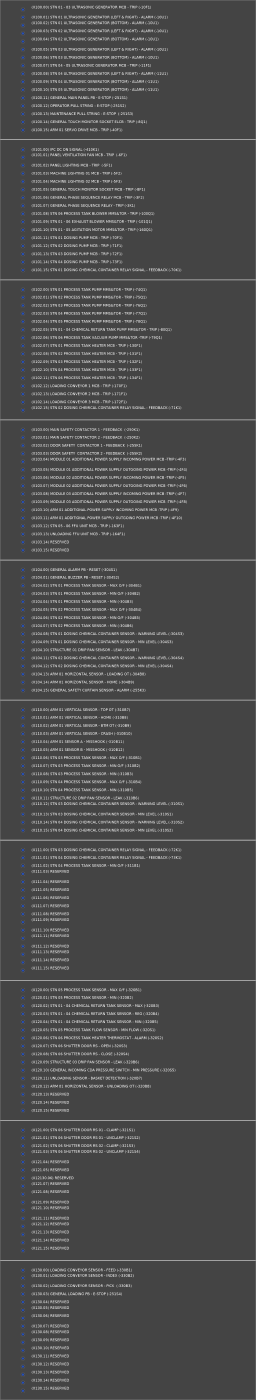
VISUALIZATION Popup_IOinput  // 733x3998
    Rectangle (0,0 733x398)
    Label (87,15 625x24), "(X100.00) STN 01 - 03 ULTRASONIC GENERATOR MCB - TRIP (-10F1)"
    Lamp1 (58,20 15x15), variable: ARbDI[eX10000_Stn01_03UltrasonicGeneratorMcb_Trip], style: Lamp-Lamp1-Blue
    Label (87,37 625x24), "(X100.01) STN 01 ULTRASONIC GENERATOR (LEFT & RIGHT) - ALARM (-10U1)"
    Lamp1 (58,42 15x15), variable: ARbDI[eX10001_Stn01UltrasonicGeneratorLeftRight_Alarm], style: Lamp-Lamp1-Blue
    Label (87,83 625x24), "(X100.03) STN 02 ULTRASONIC GENERATOR (LEFT & RIGHT) - ALARM (-10U1)"
    Lamp1 (58,88 15x15), variable: ARbDI[eX10003_Stn02UltrasonicGeneratorLeftRight_Alarm], style: Lamp-Lamp1-Blue
    Label (87,60 625x24), "(X100.02) STN 01 ULTRASONIC GENERATOR (BOTTOM) - ALARM (-10U1)"
    Lamp1 (58,65 15x15), variable: ARbDI[eX10002_Stn01UltrasonicGeneratorBottom_Alarm], style: Lamp-Lamp1-Blue
    Label (87,175 625x24), "(X100.07) STN 04 - 05 ULTRASONIC GENERATOR MCB - TRIP (-11F1)"
    Lamp1 (58,180 15x15), variable: ARbDI[eX10007_Stn04_05UltrasonicGeneratorMcb_Trip], style: Lamp-Lamp1-Blue
    Label (87,106 625x24), "(X100.04) STN 02 ULTRASONIC GENERATOR (BOTTOM) - ALARM (-10U1)"
    Lamp1 (58,111 15x15), variable: ARbDI[eX10004_Stn02UltrasonicGeneratorBottom_Alarm], style: Lamp-Lamp1-Blue
    Label (87,129 625x24), "(X100.05) STN 03 ULTRASONIC GENERATOR (LEFT & RIGHT) - ALARM (-10U1)"
    Lamp1 (58,134 15x15), variable: ARbDI[eX10005_Stn03UltrasonicGeneratorLeftRight_Alarm], style: Lamp-Lamp1-Blue
    Label (87,152 625x24), "(X100.06) STN 03 ULTRASONIC GENERATOR (BOTTOM) - ALARM (-10U1)"
    Lamp1 (58,157 15x15), variable: ARbDI[eX10006_Stn03UltrasonicGeneratorBottom_Alarm], style: Lamp-Lamp1-Blue
    Label (87,359 625x24), "(X100.15) ARM 01 SERVO DRIVE MCB - TRIP (-40F1)"
    Lamp1 (58,364 15x15), variable: ARbDI[eX10015_Arm01ServoDriveMcb_Trip], style: Lamp-Lamp1-Blue
    Label (87,198 625x24), "(X100.08) STN 04 ULTRASONIC GENERATOR (LEFT & RIGHT) - ALARM (-11U1)"
    Lamp1 (58,203 15x15), variable: ARbDI[eX10008_Stn04UltrasonicGeneratorLeftRight_Alarm], style: Lamp-Lamp1-Blue
    Label (87,221 625x24), "(X100.09) STN 04 ULTRASONIC GENERATOR (BOTTOM) - ALARM (-11U1)"
    Lamp1 (58,226 15x15), variable: ARbDI[eX10009_Stn04UltrasonicGeneratorBottom_Alarm], style: Lamp-Lamp1-Blue
    Label (87,267 625x24), "(X100.11) GENERAL MAIN PANEL PB - E-STOP (-251S1)"
    Lamp1 (58,272 15x15), variable: ARbDI[eX10011_GeneralMainPanelPb_E_Stop], style: Lamp-Lamp1-Blue
    Label (87,244 625x24), "(X100.10) STN 05 ULTRASONIC GENERATOR (BOTTOM) - ALARM (-11U1)"
    Lamp1 (58,249 15x15), variable: ARbDI[eX10010_Stn05UltrasonicGeneratorBottom_Alarm], style: Lamp-Lamp1-Blue
    Label (87,290 625x24), "(X100.12) OPERATOR PULL STRING - E-STOP (-251S2)"
    Lamp1 (58,295 15x15), variable: ARbDI[eX10012_OperatorPullString_E_Stop], style: Lamp-Lamp1-Blue
    Label (87,313 625x24), "(X100.13) MAINTENANCE PULL STRING - E-STOP (-251S3)"
    Lamp1 (58,318 15x15), variable: ARbDI[eX10013_MaintenancePullString_E_Stop], style: Lamp-Lamp1-Blue
    Label (87,336 625x24), "(X100.14) GENERAL TOUCH MONITOR SOCKET ELCB - TRIP (-8Q1)"
    Lamp1 (58,341 15x15), variable: ARbDI[eX10014_GeneralTouchMonitorSocketElcb_Trip], style: Lamp-Lamp1-Blue
    Rectangle (0,400 733x398)
    Label (87,415 625x24), "(X101.00) IPC DC ON SIGNAL (-410K1)"
    Lamp1 (58,420 15x15), variable: ARbDI[eX10100_IpcDcOnSignal], style: Lamp-Lamp1-Blue
    Label (87,437 625x24), "(X101.01) PANEL VENTILATION FAN MCB - TRIP (-6F1)"
    Lamp1 (58,442 15x15), variable: ARbDI[eX10101_PanelVentilationFanMcb_Trip], style: Lamp-Lamp1-Blue
    Label (87,483 625x24), "(X101.03) MACHINE LIGHTING 01 MCB - TRIP (-5F2)"
    Lamp1 (58,488 15x15), variable: ARbDI[eX10103_MachineLighting01Mcb_Trip], style: Lamp-Lamp1-Blue
    Label (87,460 625x24), "(X101.02) PANEL LIGHTING MCB - TRIP (-5F1)"
    Lamp1 (58,465 15x15), variable: ARbDI[eX10102_PanelLightingMcb_Trip], style: Lamp-Lamp1-Blue
    Label (87,575 625x24), "(X101.07) GENERAL PHASE SEQUENCE RELAY - TRIP (-3K1)"
    Lamp1 (58,580 15x15), variable: ARbDI[eX10107_GeneralPhaseSequenceRelay_Trip], style: Lamp-Lamp1-Blue
    Label (87,506 625x24), "(X101.04) MACHINE LIGHTING 02 MCB - TRIP (-5F3)"
    Lamp1 (58,511 15x15), variable: ARbDI[eX10104_MachineLighting02Mcb_Trip], style: Lamp-Lamp1-Blue
    Label (87,529 625x24), "(X101.05) GENERAL TOUCH MONITOR SOCKET MCB - TRIP (-8F1)"
    Lamp1 (58,534 15x15), variable: ARbDI[eX10105_GeneralTouchMonitorSocketMcb_Trip], style: Lamp-Lamp1-Blue
    Label (87,552 625x24), "(X101.06) GENERAL PHASE SEQUENCE RELAY MCB - TRIP (-3F2)"
    Lamp1 (58,557 15x15), variable: ARbDI[eX10106_GeneralPhaseSequenceRelayMcb_Trip], style: Lamp-Lamp1-Blue
    Label (87,759 625x24), "(X101.15) STN 01 DOSING CHEMICAL CONTAINER RELAY SIGNAL - FEEDBACK (-70K1)"
    Lamp1 (58,764 15x15), variable: ARbDI[eX10115_Stn01DosingChemicalContainerRelaySignal_Feedback], style: Lamp-Lamp1-Blue
    Label (87,598 625x24), "(X101.08) STN 06 PROCESS TANK BLOWER MMS&TOR - TRIP (-100Q1)"
    Lamp1 (58,603 15x15), variable: ARbDI[eX10108_Stn06ProcessTankBlowerMms_Tor_Trip], style: Lamp-Lamp1-Blue
    Label (87,621 625x24), "(X101.09) STN 01 - 06 EXHAUST BLOWER MMS&TOR - TRIP (-101Q1)"
    Lamp1 (58,626 15x15), variable: ARbDI[eX10109_Stn01_06ExhaustBlowerMms_Tor_Trip], style: Lamp-Lamp1-Blue
    Label (87,667 625x24), "(X101.11) STN 01 DOSING PUMP MCB - TRIP (-70F1)"
    Lamp1 (58,672 15x15), variable: ARbDI[eX10111_Stn01DosingPumpMcb_Trip], style: Lamp-Lamp1-Blue
    Label (87,644 625x24), "(X101.10) STN 01 - 05 AGITATION MOTOR MMS&TOR - TRIP (-160Q1)"
    Lamp1 (58,649 15x15), variable: ARbDI[eX10110_Stn01_05AgitationMotorMms_Tor_Trip], style: Lamp-Lamp1-Blue
    Label (87,690 625x24), "(X101.12) STN 02 DOSING PUMP MCB - TRIP (-71F1)"
    Lamp1 (58,695 15x15), variable: ARbDI[eX10112_Stn02DosingPumpMcb_Trip], style: Lamp-Lamp1-Blue
    Label (87,713 625x24), "(X101.13) STN 03 DOSING PUMP MCB - TRIP (-72F1)"
    Lamp1 (58,718 15x15), variable: ARbDI[eX10113_Stn03DosingPumpMcb_Trip], style: Lamp-Lamp1-Blue
    Label (87,736 625x24), "(X101.14) STN 04 DOSING PUMP MCB - TRIP (-73F1)"
    Lamp1 (58,741 15x15), variable: ARbDI[eX10114_Stn04DosingPumpMcb_Trip], style: Lamp-Lamp1-Blue
    Rectangle (0,800 733x398)
    Label (87,815 642x24), "(X102.00) STN 01 PROCESS TANK PUMP MMS&TOR - TRIP (-74Q1)"
    Lamp1 (58,820 15x15), variable: ARbDI[eX10200_Stn01ProcessTankPumpMms_Tor_Trip], style: Lamp-Lamp1-Blue
    Label (87,837 641x24), "(X102.01) STN 02 PROCESS TANK PUMP MMS&TOR - TRIP (-75Q1)"
    Lamp1 (58,842 15x15), variable: ARbDI[eX10201_Stn02ProcessTankPumpMms_Tor_Trip], style: Lamp-Lamp1-Blue
    Label (87,883 641x24), "(X102.03) STN 04 PROCESS TANK PUMP MMS&TOR - TRIP (-77Q1)"
    Lamp1 (58,888 15x15), variable: ARbDI[eX10203_Stn04ProcessTankPumpMms_Tor_Trip], style: Lamp-Lamp1-Blue
    Label (87,860 643x24), "(X102.02) STN 03 PROCESS TANK PUMP MMS&TOR - TRIP (-76Q1)"
    Lamp1 (58,865 15x15), variable: ARbDI[eX10202_Stn03ProcessTankPumpMms_Tor_Trip], style: Lamp-Lamp1-Blue
    Label (87,975 625x24), "(X102.07) STN 01 PROCESS TANK HEATER MCB - TRIP (-130F1)"
    Lamp1 (58,980 15x15), variable: ARbDI[eX10207_Stn01ProcessTankHeaterMcb_Trip], style: Lamp-Lamp1-Blue
    Label (87,906 641x24), "(X102.04) STN 05 PROCESS TANK PUMP MMS&TOR - TRIP (-78Q1)"
    Lamp1 (58,911 15x15), variable: ARbDI[eX10204_Stn05ProcessTankPumpMms_Tor_Trip], style: Lamp-Lamp1-Blue
    Label (87,929 642x24), "(X102.05) STN 01 - 04 CHEMICAL RETURN TANK PUMP MMS&TOR - TRIP (-80Q1)"
    Lamp1 (58,934 15x15), variable: ARbDI[eX10205_Stn01_04ChemicalReturnTankPumpMms_Tor_Trip], style: Lamp-Lamp1-Blue
    Label (87,952 642x24), "(X102.06) STN 06 PROCESS TANK VACUUM PUMP MMS&TOR -TRIP (-79Q1)"
    Lamp1 (58,957 15x15), variable: ARbDI[eX10206_Stn06ProcessTankVacuumPumpMms_Tor_Trip], style: Lamp-Lamp1-Blue
    Label (87,1159 625x24), "(X102.15) STN 02 DOSING CHEMICAL CONTAINER RELAY SIGNAL - FEEDBACK (-71K1)"
    Lamp1 (58,1164 15x15), variable: ARbDI[eX10215_Stn02DosingChemicalContainerRelaySignal_Feedback], style: Lamp-Lamp1-Blue
    Label (87,998 625x24), "(X102.08) STN 02 PROCESS TANK HEATER MCB - TRIP (-131F1)"
    Lamp1 (58,1003 15x15), variable: ARbDI[eX10208_Stn02ProcessTankHeaterMcb_Trip], style: Lamp-Lamp1-Blue
    Label (87,1021 625x24), "(X102.09) STN 03 PROCESS TANK HEATER MCB - TRIP (-132F1)"
    Lamp1 (58,1026 15x15), variable: ARbDI[eX10209_Stn03ProcessTankHeaterMcb_Trip], style: Lamp-Lamp1-Blue
    Label (87,1067 625x24), "(X102.11) STN 06 PROCESS TANK HEATER MCB - TRIP (-134F1)"
    Lamp1 (58,1072 15x15), variable: ARbDI[eX10211_Stn06ProcessTankHeaterMcb_Trip], style: Lamp-Lamp1-Blue
    Label (87,1044 625x24), "(X102.10) STN 04 PROCESS TANK HEATER MCB - TRIP (-133F1)"
    Lamp1 (58,1049 15x15), variable: ARbDI[eX10210_Stn04ProcessTankHeaterMcb_Trip], style: Lamp-Lamp1-Blue
    Label (87,1090 625x24), "(X102.12) LOADING CONVEYOR 1 MCB - TRIP (-170F1)"
    Lamp1 (58,1095 15x15), variable: ARbDI[eX10212_LoadingConveyor1Mcb_Trip], style: Lamp-Lamp1-Blue
    Label (87,1113 625x24), "(X102.13) LOADING CONVEYOR 2 MCB - TRIP (-171F1)"
    Lamp1 (58,1118 15x15), variable: ARbDI[eX10213_LoadingConveyor2Mcb_Trip], style: Lamp-Lamp1-Blue
    Label (87,1136 625x24), "(X102.14) LOADING CONVEYOR 3 MCB - TRIP (-172F1)"
    Lamp1 (58,1141 15x15), variable: ARbDI[eX10214_LoadingConveyor3Mcb_Trip], style: Lamp-Lamp1-Blue
    Rectangle (0,1600 733x398)
    Label (87,1615 625x24), "(X104.00) GENERAL ALARM PB - RESET (-304S1)"
    Lamp1 (58,1620 15x15), variable: ARbDI[eX10400_GeneralAlarmPb_Reset], style: Lamp-Lamp1-Blue
    Label (87,1637 625x24), "(X104.01) GENERAL BUZZER PB - RESET (-304S2)"
    Lamp1 (58,1642 15x15), variable: ARbDI[eX10401_GeneralBuzzerPb_Reset], style: Lamp-Lamp1-Blue
    Label (87,1683 625x24), "(X104.03) STN 01 PROCESS TANK SENSOR - MIN O/F (-304B2)"
    Lamp1 (58,1688 15x15), variable: ARbDI[eX10403_Stn01ProcessTankSensor_MinOverflow], style: Lamp-Lamp1-Blue
    Label (87,1660 625x24), "(X104.02) STN 01 PROCESS TANK SENSOR - MAX O/F (-304B1)"
    Lamp1 (58,1665 15x15), variable: ARbDI[eX10402_Stn01ProcessTankSensor_MaxOverflow], style: Lamp-Lamp1-Blue
    Label (87,1775 625x24), "(X104.07) STN 02 PROCESS TANK SENSOR - MIN (-304B6)"
    Lamp1 (58,1780 15x15), variable: ARbDI[eX10407_Stn02ProcessTankSensor_Min], style: Lamp-Lamp1-Blue
    Label (87,1706 625x24), "(X104.04) STN 01 PROCESS TANK SENSOR - MIN (-304B3)"
    Lamp1 (58,1711 15x15), variable: ARbDI[eX10404_Stn01ProcessTankSensor_Min], style: Lamp-Lamp1-Blue
    Label (87,1729 625x24), "(X104.05) STN 02 PROCESS TANK SENSOR - MAX O/F (-304B4)"
    Lamp1 (58,1734 15x15), variable: ARbDI[eX10405_Stn02ProcessTankSensor_MaxOverflow], style: Lamp-Lamp1-Blue
    Label (87,1752 625x24), "(X104.06) STN 02 PROCESS TANK SENSOR - MIN O/F (-304B5)"
    Lamp1 (58,1757 15x15), variable: ARbDI[eX10406_Stn02ProcessTankSensor_MinOverflow], style: Lamp-Lamp1-Blue
    Label (87,1959 625x24), "(X104.15) GENERAL SAFETY CURTAIN SENSOR - ALARM (-255K3)"
    Lamp1 (58,1964 15x15), variable: ARbDI[eX10415_GeneralSafetyCurtainSensor_Alarm], style: Lamp-Lamp1-Blue
    Label (87,1798 625x24), "(X104.08) STN 01 DOSING CHEMICAL CONTAINER SENSOR - WARNING LEVEL (-304S3)"
    Lamp1 (58,1803 15x15), variable: ARbDI[eX10408_Stn01DosingChemicalContainerSensor_WarningLevel], style: Lamp-Lamp1-Blue
    Label (87,1821 625x24), "(X104.09) STN 01 DOSING CHEMICAL CONTAINER SENSOR - MIN LEVEL (-304S3)"
    Lamp1 (58,1826 15x15), variable: ARbDI[eX10409_Stn01DosingChemicalContainerSensor_MinLevel], style: Lamp-Lamp1-Blue
    Label (87,1867 625x24), "(X104.11) STN 02 DOSING CHEMICAL CONTAINER SENSOR - WARNING LEVEL (-304S4)"
    Lamp1 (58,1872 15x15), variable: ARbDI[eX10411_Stn02DosingChemicalContainerSensor_WarningLevel], style: Lamp-Lamp1-Blue
    Label (87,1844 625x24), "(X104.10) STRUCTURE 01 DRIP PAN SENSOR - LEAK (-304B7)"
    Lamp1 (58,1849 15x15), variable: ARbDI[eX10410_Structure01DripPanSensor_Leak], style: Lamp-Lamp1-Blue
    Label (87,1890 625x24), "(X104.12) STN 02 DOSING CHEMICAL CONTAINER SENSOR - MIN LEVEL (-304S4)"
    Lamp1 (58,1895 15x15), variable: ARbDI[eX10412_Stn02DosingChemicalContainerSensor_MinLevel], style: Lamp-Lamp1-Blue
    Label (87,1913 625x24), "(X104.13) ARM 01 HORIZONTAL SENSOR - LOADING OT (-304B8)"
    Lamp1 (58,1918 15x15), variable: ARbDI[eX10413_Arm01HorizontalSensor_LoadingOt], style: Lamp-Lamp1-Blue
    Label (87,1936 625x24), "(X104.14) ARM 01 HORIZONTAL SENSOR - HOME (-304B9)"
    Lamp1 (58,1941 15x15), variable: ARbDI[eX10414_Arm01HorizontalSensor_Home], style: Lamp-Lamp1-Blue
    Rectangle (0,1200 733x398)
    Label (87,1215 625x24), "(X103.00) MAIN SAFETY CONTACTOR 1 - FEEDBACK (-250K1)"
    Lamp1 (58,1220 15x15), variable: ARbDI[eX10300_MainSafetyContactor1_Feedback], style: Lamp-Lamp1-Blue
    Label (87,1237 625x24), "(X103.01) MAIN SAFETY CONTACTOR 2 - FEEDBACK (-250K2)"
    Lamp1 (58,1242 15x15), variable: ARbDI[eX10301_MainSafetyContactor2_Feedback], style: Lamp-Lamp1-Blue
    Label (87,1283 625x24), "(X103.03) DOOR SAFETY CONTACTOR 2 - FEEDBACK (-255K2)"
    Lamp1 (58,1288 15x15), variable: ARbDI[eX10303_DoorSafetyContactor2_Feedback], style: Lamp-Lamp1-Blue
    Label (87,1260 625x24), "(X103.02) DOOR SAFETY CONTACTOR 1 - FEEDBACK (-255K1)"
    Lamp1 (58,1265 15x15), variable: ARbDI[eX10302_DoorSafetyContactor1_Feedback], style: Lamp-Lamp1-Blue
    Label (87,1375 625x24), "(X103.07) MODULE 02 ADDITIONAL POWER SUPPLY OUTGOING POWER MCB -TRIP (-4F6)"
    Lamp1 (58,1380 15x15), variable: ARbDI[eX10307_Module02AdditionalPowerSupplyOutgoingPowerMcb_Trip], style: Lamp-Lamp1-Blue
    Label (87,1306 625x24), "(X103.04) MODULE 01 ADDITIONAL POWER SUPPLY INCOMING POWER MCB -TRIP (-4F3)"
    Lamp1 (58,1311 15x15), variable: ARbDI[eX10304_Module01AdditionalPowerSupplyIncomingPowerMcb_Trip], style: Lamp-Lamp1-Blue
    Label (87,1329 625x24), "(X103.05) MODULE 01 ADDITIONAL POWER SUPPLY OUTGOING POWER MCB -TRIP (-4F4)"
    Lamp1 (58,1334 15x15), variable: ARbDI[eX10305_Module01AdditionalPowerSupplyOutgoingPowerMcb_Trip], style: Lamp-Lamp1-Blue
    Label (87,1352 625x24), "(X103.06) MODULE 02 ADDITIONAL POWER SUPPLY INCOMING POWER MCB -TRIP (-4F5)"
    Lamp1 (58,1357 15x15), variable: ARbDI[eX10306_Module02AdditionalPowerSupplyIncomingPowerMcb_Trip], style: Lamp-Lamp1-Blue
    Label (87,1559 625x24), "(X103.15) RESERVED"
    Lamp1 (58,1564 15x15), variable: ARbDI[eX10315_Reserved], style: Lamp-Lamp1-Blue
    Label (87,1398 625x24), "(X103.08) MODULE 03 ADDITIONAL POWER SUPPLY INCOMING POWER MCB -TRIP (-4F7)"
    Lamp1 (58,1403 15x15), variable: ARbDI[eX10308_Module03AdditionalPowerSupplyIncomingPowerMcb_Trip], style: Lamp-Lamp1-Blue
    Label (87,1421 625x24), "(X103.09) MODULE 03 ADDITIONAL POWER SUPPLY OUTGOING POWER MCB -TRIP (-4F8)"
    Lamp1 (58,1426 15x15), variable: ARbDI[eX10309_Module03AdditionalPowerSupplyOutgoingPowerMcb_Trip], style: Lamp-Lamp1-Blue
    Label (87,1467 625x24), "(X103.11) ARM 01 ADDITIONAL POWER SUPPLY OUTGOING POWER MCB -TRIP (-4F10)"
    Lamp1 (58,1472 15x15), variable: ARbDI[eX10311_Arm01AdditionalPowerSupplyOutgoingPowerMcb_Trip], style: Lamp-Lamp1-Blue
    Label (87,1444 625x24), "(X103.10) ARM 01 ADDITIONAL POWER SUPPLY INCOMING POWER MCB -TRIP (-4F9)"
    Lamp1 (58,1449 15x15), variable: ARbDI[eX10310_Arm01AdditionalPowerSupplyIncomingPowerMcb_Trip], style: Lamp-Lamp1-Blue
    Label (87,1490 625x24), "(X103.12) STN 05 - 06 FFU UNIT MCB - TRIP (-163F1)"
    Lamp1 (58,1495 15x15), variable: ARbDI[eX10312_Stn05_06FfuUnitMcb_Trip], style: Lamp-Lamp1-Blue
    Label (87,1513 625x24), "(X103.13) UNLOADING FFU UNIT MCB - TRIP (-164F1)"
    Lamp1 (58,1518 15x15), variable: ARbDI[eX10313_UnloadingFfuUnitMcb_Trip], style: Lamp-Lamp1-Blue
    Label (87,1536 625x24), "(X103.14) RESERVED"
    Lamp1 (58,1541 15x15), variable: ARbDI[eX10314_Reserved], style: Lamp-Lamp1-Blue
    Rectangle (0,2000 733x398)
    Label (87,2015 625x24), "(X110.00) ARM 01 VERTICAL SENSOR - TOP OT (-310B7)"
    Lamp1 (58,2020 15x15), variable: ARbDI[eX11000_Arm01VerticalSensor_TopOt], style: Lamp-Lamp1-Blue
    Label (87,2037 625x24), "(X110.01) ARM 01 VERTICAL SENSOR - HOME (-310B8)"
    Lamp1 (58,2042 15x15), variable: ARbDI[eX11001_Arm01VerticalSensor_Home], style: Lamp-Lamp1-Blue
    Label (87,2083 625x24), "(X110.03) ARM 01 VERTICAL SENSOR - CRASH (-310B10)"
    Lamp1 (58,2088 15x15), variable: ARbDI[eX11003_Arm01VerticalSensor_Crash], style: Lamp-Lamp1-Blue
    Label (87,2060 625x24), "(X110.02) ARM 01 VERTICAL SENSOR - BTM OT (-310B9)"
    Lamp1 (58,2065 15x15), variable: ARbDI[eX11002_Arm01VerticalSensor_BtmOt], style: Lamp-Lamp1-Blue
    Label (87,2175 625x24), "(X110.07) STN 03 PROCESS TANK SENSOR - MIN O/F (-310B2)"
    Lamp1 (58,2180 15x15), variable: ARbDI[eX11007_Stn03ProcessTankSensor_MinOverflow], style: Lamp-Lamp1-Blue
    Label (87,2106 625x24), "(X110.04) ARM 01 SENSOR A - MISSHOOK (-310B11)"
    Lamp1 (58,2111 15x15), variable: ARbDI[eX11004_Arm01SensorA_Misshook], style: Lamp-Lamp1-Blue
    Label (87,2129 625x24), "(X110.05) ARM 01 SENSOR B - MISSHOOK (-310B12)"
    Lamp1 (58,2134 15x15), variable: ARbDI[eX11005_Arm01SensorB_Misshook], style: Lamp-Lamp1-Blue
    Label (87,2152 625x24), "(X110.06) STN 03 PROCESS TANK SENSOR - MAX O/F (-310B1)"
    Lamp1 (58,2157 15x15), variable: ARbDI[eX11006_Stn03ProcessTankSensor_MaxOverflow], style: Lamp-Lamp1-Blue
    Label (87,2359 625x24), "(X110.15) STN 04 DOSING CHEMICAL CONTAINER SENSOR - MIN LEVEL (-310S2)"
    Lamp1 (58,2364 15x15), variable: ARbDI[eX11015_Stn04DosingChemicalContainerSensor_MinLevel], style: Lamp-Lamp1-Blue
    Label (87,2198 625x24), "(X110.08) STN 03 PROCESS TANK SENSOR - MIN (-310B3)"
    Lamp1 (58,2203 15x15), variable: ARbDI[eX11008_Stn03ProcessTankSensor_Min], style: Lamp-Lamp1-Blue
    Label (87,2221 625x24), "(X110.09) STN 04 PROCESS TANK SENSOR - MAX O/F (-310B4)"
    Lamp1 (58,2226 15x15), variable: ARbDI[eX11009_Stn04ProcessTankSensor_MaxOverflow], style: Lamp-Lamp1-Blue
    Label (87,2267 625x24), "(X110.11) STRUCTURE 02 DRIP PAN SENSOR - LEAK (-310B6)"
    Lamp1 (58,2272 15x15), variable: ARbDI[eX11011_Structure02DripPanSensor_Leak], style: Lamp-Lamp1-Blue
    Label (87,2244 625x24), "(X110.10) STN 04 PROCESS TANK SENSOR - MIN (-310B5)"
    Lamp1 (58,2249 15x15), variable: ARbDI[eX11010_Stn04ProcessTankSensor_Min], style: Lamp-Lamp1-Blue
    Label (87,2290 625x24), "(X110.12) STN 03 DOSING CHEMICAL CONTAINER SENSOR - WARNING LEVEL (-310S1)"
    Lamp1 (58,2295 15x15), variable: ARbDI[eX11012_Stn03DosingChemicalContainerSensor_WarningLevel], style: Lamp-Lamp1-Blue
    Label (87,2313 625x24), "(X110.13) STN 03 DOSING CHEMICAL CONTAINER SENSOR - MIN LEVEL (-310S1)"
    Lamp1 (58,2318 15x15), variable: ARbDI[eX11013_Stn03DosingChemicalContainerSensor_MinLevel], style: Lamp-Lamp1-Blue
    Label (87,2336 625x24), "(X110.14) STN 04 DOSING CHEMICAL CONTAINER SENSOR - WARNING LEVEL (-310S2)"
    Lamp1 (58,2341 15x15), variable: ARbDI[eX11014_Stn04DosingChemicalContainerSensor_WarningLevel], style: Lamp-Lamp1-Blue
    Rectangle (0,2400 733x398)
    Label (87,2415 625x24), "(X111.00) STN 03 DOSING CHEMICAL CONTAINER RELAY SIGNAL - FEEDBACK (-72K1)"
    Lamp1 (58,2420 15x15), variable: ARbDI[eX11100_Stn03DosingChemicalContainerRelaySignal_Feedback], style: Lamp-Lamp1-Blue
    Label (87,2437 625x24), "(X111.01) STN 04 DOSING CHEMICAL CONTAINER RELAY SIGNAL - FEEDBACK (-73K1)"
    Lamp1 (58,2442 15x15), variable: ARbDI[eX11101_Stn04DosingChemicalContainerRelaySignal_Feedback], style: Lamp-Lamp1-Blue
    Label (87,2483 625x24), "(X111.03) RESERVED"
    Lamp1 (58,2488 15x15), variable: ARbDI[eX11103_Reserved], style: Lamp-Lamp1-Blue
    Label (87,2460 625x24), "(X111.02) STN 04 PROCESS TANK SENSOR - MIN O/F (-311B1)"
    Lamp1 (58,2465 15x15), variable: ARbDI[eX11102_Stn04ProcessTankSensor_MinOverflow], style: Lamp-Lamp1-Blue
    Label (87,2575 625x24), "(X111.07) RESERVED"
    Lamp1 (58,2580 15x15), variable: ARbDI[eX11107_Reserved], style: Lamp-Lamp1-Blue
    Label (87,2506 625x24), "(X111.04) RESERVED"
    Lamp1 (58,2511 15x15), variable: ARbDI[eX11104_Reserved], style: Lamp-Lamp1-Blue
    Label (87,2529 625x24), "(X111.05) RESERVED"
    Lamp1 (58,2534 15x15), variable: ARbDI[eX11105_Reserved], style: Lamp-Lamp1-Blue
    Label (87,2552 625x24), "(X111.06) RESERVED"
    Lamp1 (58,2557 15x15), variable: ARbDI[eX11106_Reserved], style: Lamp-Lamp1-Blue
    Label (87,2759 625x24), "(X111.15) RESERVED"
    Lamp1 (58,2764 15x15), variable: ARbDI[eX11115_Reserved], style: Lamp-Lamp1-Blue
    Label (87,2598 625x24), "(X111.08) RESERVED"
    Lamp1 (58,2603 15x15), variable: ARbDI[eX11108_Reserved], style: Lamp-Lamp1-Blue
    Label (87,2621 625x24), "(X111.09) RESERVED"
    Lamp1 (58,2626 15x15), variable: ARbDI[eX11109_Reserved], style: Lamp-Lamp1-Blue
    Label (87,2667 625x24), "(X111.11) RESERVED"
    Lamp1 (58,2672 15x15), variable: ARbDI[eX11111_Reserved], style: Lamp-Lamp1-Blue
    Label (87,2644 625x24), "(X111.10) RESERVED"
    Lamp1 (58,2649 15x15), variable: ARbDI[eX11110_Reserved], style: Lamp-Lamp1-Blue
    Label (87,2690 625x24), "(X111.12) RESERVED"
    Lamp1 (58,2695 15x15), variable: ARbDI[eX11112_Reserved], style: Lamp-Lamp1-Blue
    Label (87,2713 625x24), "(X111.13) RESERVED"
    Lamp1 (58,2718 15x15), variable: ARbDI[eX11113_Reserved], style: Lamp-Lamp1-Blue
    Label (87,2736 625x24), "(X111.14) RESERVED"
    Lamp1 (58,2741 15x15), variable: ARbDI[eX11114_Reserved], style: Lamp-Lamp1-Blue
    Rectangle (0,2800 733x398)
    Label (87,2815 625x24), "(X120.00) STN 05 PROCESS TANK SENSOR - MAX O/F (-320B1)"
    Lamp1 (58,2820 15x15), variable: ARbDI[eX12000_Stn05ProcessTankSensor_MaxOverflow], style: Lamp-Lamp1-Blue
    Label (87,2837 625x24), "(X120.01) STN 05 PROCESS TANK SENSOR - MIN (-320B2)"
    Lamp1 (58,2842 15x15), variable: ARbDI[eX12001_Stn05ProcessTankSensor_Min], style: Lamp-Lamp1-Blue
    Label (87,2883 625x24), "(X120.03) STN 01 - 04 CHEMICAL RETURN TANK SENSOR - REG (-320B4)"
    Lamp1 (58,2888 15x15), variable: ARbDI[eX12003_Stn01_04ChemicalReturnTankSensor_Reg], style: Lamp-Lamp1-Blue
    Label (87,2860 625x24), "(X120.02) STN 01 - 04 CHEMICAL RETURN TANK SENSOR - MAX (-320B3)"
    Lamp1 (58,2865 15x15), variable: ARbDI[eX12002_Stn01_04ChemicalReturnTankSensor_Max], style: Lamp-Lamp1-Blue
    Label (87,2975 625x24), "(X120.07) STN 06 SHUTTER DOOR RS - OPEN (-320S3)"
    Lamp1 (58,2980 15x15), variable: ARbDI[eX12007_Stn06SlidingDoorRs_Open], style: Lamp-Lamp1-Blue
    Label (87,2906 625x24), "(X120.04) STN 01 - 04 CHEMICAL RETURN TANK SENSOR - MIN (-320B5)"
    Lamp1 (58,2911 15x15), variable: ARbDI[eX12004_Stn01_04ChemicalReturnTankSensor_Min], style: Lamp-Lamp1-Blue
    Label (87,2929 625x24), "(X120.05) STN 05 PROCESS TANK FLOW SENSOR - MIN FLOW (-320S1)"
    Lamp1 (58,2934 15x15), variable: ARbDI[eX12005_Stn05ProcessTankFlowSensor_MinFlow], style: Lamp-Lamp1-Blue
    Label (87,2952 625x24), "(X120.06) STN 06 PROCESS TANK HEATER THERMOSTAT - ALARM (-320S2)"
    Lamp1 (58,2957 15x15), variable: ARbDI[eX12006_Stn06ProcessTankHeaterThermostat_Alarm], style: Lamp-Lamp1-Blue
    Label (87,3159 625x24), "(X120.15) RESERVED"
    Lamp1 (58,3164 15x15), variable: ARbDI[eX11115_Reserved], style: Lamp-Lamp1-Blue
    Label (87,2998 625x24), "(X120.08) STN 06 SHUTTER DOOR RS - CLOSE (-320S4)"
    Lamp1 (58,3003 15x15), variable: ARbDI[eX12008_Stn06SlidingDoorRs_Close], style: Lamp-Lamp1-Blue
    Label (87,3021 625x24), "(X120.09) STRUCTURE 03 DRIP PAN SENSOR - LEAK (-320B6)"
    Lamp1 (58,3026 15x15), variable: ARbDI[eX12009_Structure03DripPanSensor_Leak], style: Lamp-Lamp1-Blue
    Label (87,3067 625x24), "(X120.11) UNLOADING SENSOR - BASKET DETECTION (-320B7)"
    Lamp1 (58,3072 15x15), variable: ARbDI[eX12011_UnloadingSensor_BasketDetection], style: Lamp-Lamp1-Blue
    Label (87,3044 625x24), "(X120.10) GENERAL INCOMING CDA PRESSURE SWITCH - MIN PRESSURE (-320S5)"
    Lamp1 (58,3049 15x15), variable: ARbDI[eX12010_GeneralIncomingCdaPressureSwitch_MinPressure], style: Lamp-Lamp1-Blue
    Label (87,3090 625x24), "(X120.12) ARM 01 HORIZONTAL SENSOR - UNLOADING OT (-320B8)"
    Lamp1 (58,3095 15x15), variable: ARbDI[eX12012_Arm01HorizontalSensor_UnloadingOt], style: Lamp-Lamp1-Blue
    Label (87,3113 625x24), "(X120.13) RESERVED"
    Lamp1 (58,3118 15x15), variable: ARbDI[eX12013_Reserved], style: Lamp-Lamp1-Blue
    Label (87,3136 625x24), "(X120.14) RESERVED"
    Lamp1 (58,3141 15x15), variable: ARbDI[eX12014_Reserved], style: Lamp-Lamp1-Blue
    Rectangle (0,3600 733x398)
    Label (87,3615 625x24), "(X130.00) LOADING CONVEYOR SENSOR - FEED (-330B1)"
    Lamp1 (58,3620 15x15), variable: ARbDI[eX13000_LoadingConveyorSensor_Feed], style: Lamp-Lamp1-Blue
    Label (87,3637 625x24), "(X130.01) LOADING CONVEYOR SENSOR - INDEX (-330B2)"
    Lamp1 (58,3642 15x15), variable: ARbDI[eX13001_LoadingConveyorSensor_Index], style: Lamp-Lamp1-Blue
    Label (87,3683 625x24), "(X130.03) GENERAL LOADING PB - E-STOP (-251S4)"
    Lamp1 (58,3688 15x15), variable: ARbDI[eX13002_LoadingConveyorSensor_Pick], style: Lamp-Lamp1-Blue
    Label (87,3660 625x24), "(X130.02) LOADING CONVEYOR SENSOR - PICK (-330B3)"
    Lamp1 (58,3665 15x15), variable: ARbDI[eX13002_LoadingConveyorSensor_Pick], style: Lamp-Lamp1-Blue
    Label (87,3775 625x24), "(X130.07) RESERVED"
    Lamp1 (58,3780 15x15), variable: ARbDI[eX13006_Reserved], style: Lamp-Lamp1-Blue
    Label (87,3706 625x24), "(X130.04) RESERVED"
    Lamp1 (58,3711 15x15), variable: ARbDI[eX13003_GeneralLoadingPb_E_Stop], style: Lamp-Lamp1-Blue
    Label (87,3729 625x24), "(X130.05) RESERVED"
    Lamp1 (58,3734 15x15), variable: ARbDI[eX13004_Reserved], style: Lamp-Lamp1-Blue
    Label (87,3752 625x24), "(X130.06) RESERVED"
    Lamp1 (58,3757 15x15), variable: ARbDI[eX13005_Reserved], style: Lamp-Lamp1-Blue
    Label (87,3959 625x24), "(X130.15) RESERVED"
    Lamp1 (58,3964 15x15), variable: ARbDI[eX13015_Reserved], style: Lamp-Lamp1-Blue
    Label (87,3798 625x24), "(X130.08) RESERVED"
    Lamp1 (58,3803 15x15), variable: ARbDI[eX13007_Reserved], style: Lamp-Lamp1-Blue
    Label (87,3821 625x24), "(X130.09) RESERVED"
    Lamp1 (58,3826 15x15), variable: ARbDI[eX13008_Reserved], style: Lamp-Lamp1-Blue
    Label (87,3867 625x24), "(X130.11) RESERVED"
    Lamp1 (58,3872 15x15), variable: ARbDI[eX13011_Reserved], style: Lamp-Lamp1-Blue
    Label (87,3844 625x24), "(X130.10) RESERVED"
    Lamp1 (58,3849 15x15), variable: ARbDI[eX13009_Reserved], style: Lamp-Lamp1-Blue
    Label (87,3890 625x24), "(X130.12) RESERVED"
    Lamp1 (58,3895 15x15), variable: ARbDI[eX13012_Reserved], style: Lamp-Lamp1-Blue
    Label (87,3913 625x24), "(X130.13) RESERVED"
    Lamp1 (58,3918 15x15), variable: ARbDI[eX13013_Reserved], style: Lamp-Lamp1-Blue
    Label (87,3936 625x24), "(X130.14) RESERVED"
    Lamp1 (58,3941 15x15), variable: ARbDI[eX13014_Reserved], style: Lamp-Lamp1-Blue
    Rectangle (0,3200 733x398)
    Label (87,3215 625x24), "(X121.00) STN 06 SHUTTER DOOR RS 01 - CLAMP (-321S1)"
    Lamp1 (58,3220 15x15), variable: ARbDI[eX12100_Stn06SlidingDoorRs01_Clamp], style: Lamp-Lamp1-Blue
    Label (87,3237 625x24), "(X121.01) STN 06 SHUTTER DOOR RS 01 - UNCLAMP (-321S2)"
    Lamp1 (58,3242 15x15), variable: ARbDI[eX12101_Stn06SlidingDoorRs01_Unclamp], style: Lamp-Lamp1-Blue
    Label (87,3283 625x24), "(X121.03) STN 06 SHUTTER DOOR RS 02 - UNCLAMP (-321S4)"
    Lamp1 (58,3288 15x15), variable: ARbDI[eX12103_Stn06SlidingDoorRs02_Unclamp], style: Lamp-Lamp1-Blue
    Label (87,3260 625x24), "(X121.02) STN 06 SHUTTER DOOR RS 02 - CLAMP (-321S3)"
    Lamp1 (58,3265 15x15), variable: ARbDI[eX12102_Stn06SlidingDoorRs02_Clamp], style: Lamp-Lamp1-Blue
    Label (87,3375 625x24), "(X121.07) RESERVED"
    Lamp1 (58,3380 15x15), variable: ARbDI[eX12107_Reserved], style: Lamp-Lamp1-Blue
    Label (87,3306 625x24), "(X121.04) RESERVED"
    Lamp1 (58,3311 15x15), variable: ARbDI[eX12104_Reserved], style: Lamp-Lamp1-Blue
    Label (87,3329 625x24), "(X121.05) RESERVED"
    Lamp1 (58,3334 15x15), variable: ARbDI[eX12105_Reserved], style: Lamp-Lamp1-Blue
    Label (87,3352 625x24), "(X12130.06) RESERVED"
    Lamp1 (58,3357 15x15), variable: ARbDI[eX12106_Reserved], style: Lamp-Lamp1-Blue
    Label (87,3559 625x24), "(X121.15) RESERVED"
    Lamp1 (58,3564 15x15), variable: ARbDI[eX12115_Reserved], style: Lamp-Lamp1-Blue
    Label (87,3398 625x24), "(X121.08) RESERVED"
    Lamp1 (58,3403 15x15), variable: ARbDI[eX12108_Reserved], style: Lamp-Lamp1-Blue
    Label (87,3421 625x24), "(X121.09) RESERVED"
    Lamp1 (58,3426 15x15), variable: ARbDI[eX12109_Reserved], style: Lamp-Lamp1-Blue
    Label (87,3467 625x24), "(X121.11) RESERVED"
    Lamp1 (58,3472 15x15), variable: ARbDI[eX12111_Reserved], style: Lamp-Lamp1-Blue
    Label (87,3444 625x24), "(X121.10) RESERVED"
    Lamp1 (58,3449 15x15), variable: ARbDI[eX12110_Reserved], style: Lamp-Lamp1-Blue
    Label (87,3490 625x24), "(X121.12) RESERVED"
    Lamp1 (58,3495 15x15), variable: ARbDI[eX12112_Reserved], style: Lamp-Lamp1-Blue
    Label (87,3513 625x24), "(X121.13) RESERVED"
    Lamp1 (58,3518 15x15), variable: ARbDI[eX12113_Reserved], style: Lamp-Lamp1-Blue
    Label (87,3536 625x24), "(X121.14) RESERVED"
    Lamp1 (58,3541 15x15), variable: ARbDI[eX12114_Reserved], style: Lamp-Lamp1-Blue
END_VISUALIZATION

(* stored: Version 1.1.0.1, ProductVersion 3.1.4024.12
   Visu Popup_IOinput: Id {61f848af-0395-4a6b-9b12-5841de9d108d} *)
